(* Logix 5000 project; controller ODSI_Testing vendor 1 type 14 code 151 rev 20.19; software revision 20.05; part 2 of 2 *)
(* tags used below, declared in another part *)
   HMI_Stop_B9 : BOOL;   // Stop PB on HMI
   ODSI_Fail_Sample1_B9 : ALIAS FOR Local:6:I.Data.8;   // ODSI sent a fail signal for sample 1
   ODSI_Fail_Sample2_B9 : ALIAS FOR Local:6:I.Data.10;   // ODSI sent a fail signal for sample 2
   ODSI_Fail_Sample3_B9 : ALIAS FOR Local:6:I.Data.12;   // ODSI sent a fail signal for sample 3
   ODSI_Pass_Sample1_B9 : ALIAS FOR Local:6:I.Data.7;   // ODSI sent a pass signal for sample 1
   ODSI_Pass_Sample2_B9 : ALIAS FOR Local:6:I.Data.9;   // ODSI sent a pass signal for sample 2
   ODSI_Pass_Sample3_B9 : ALIAS FOR Local:6:I.Data.11;   // ODSI sent a pass signal for sample 3
   ODSI_Valve1_B9 : ALIAS FOR Local:6:I.Data.4;   // ODSI requests to open valve 1
   ODSI_Valve2_B9 : ALIAS FOR Local:6:I.Data.5;   // ODSI requests to open valve 2
   ODSI_Valve3_B9 : ALIAS FOR Local:6:I.Data.6;   // ODSI requests to open valve 3
   RandomDelay : DINT;   // Random number generator 0-19
   RNG_Delay_Active_B9 : BOOL;   // HMI PB randomizing valve open delay
   S1_B9_10s_Timer : TIMER;   // Releases "ACQC in" signal after 10 seconds
   S1_PB_Input_B9 : BOOL;   // HMI PB requesting sample 1
   S1_Request_B9 : ALIAS FOR Local:5:O.Data.8;   // Output to ODSI to request Sample 1
   S2_B9_10s_Timer : TIMER;   // Releases "ACQC in" signal after 10 seconds
   S2_PB_Input_B9 : BOOL;   // HMI PB requesting sample 2
   S2_Request_B9 : ALIAS FOR Local:5:O.Data.9;   // Output to ODSI to request Sample 2
   S3_B9_10s_Timer : TIMER;   // Releases "ACQC in" signal after 10 seconds
   S3_PB_Input_B9 : BOOL;   // HMI PB requesting sample 3
   S3_Request_B9 : ALIAS FOR Local:5:O.Data.10;   // Output to ODSI to request Sample 3
   System_Running_B9 : ALIAS FOR Local:6:I.Data.3;   // ODSI signal that indicates the system is currently analyzing a sample
   Valve1_Open_B9 : ALIAS FOR Local:5:O.Data.11;   // Output to ODSI confirming valve 1 is open
   Valve1_Open_Delay_B9 : TIMER;   // Delay after Request is Initiated from ODSI
   Valve1_Open_Random_Delay_B9 : TIMER;   // Randomized delay after request for valve position is received from ODSI
   Valve2_Open_B9 : ALIAS FOR Local:5:O.Data.12;   // Output to ODSI confirming valve 2 is open
   Valve2_Open_Delay_B9 : TIMER;   // Delay after Request is Initiated from ODSI
   Valve2_Open_Random_Delay_B9 : TIMER;   // Randomized delay after request for valve position is received from ODSI
   Valve3_Open_B9 : ALIAS FOR Local:5:O.Data.13;   // Output to ODSI confirming valve 3 is open
   Valve3_Open_Delay_B9 : TIMER;   // Delay after Request is Initiated from ODSI
   Valve3_Open_Random_Delay_B9 : TIMER;   // Randomized delay after request for valve position is received from ODSI
   Valve_Block_B9 : BOOL;   // HMI PB to prevent valves from opening
   Valve_Delay_B9 : DINT;
(* MainProgram, continued *)

ROUTINE Remote_B9   (* ladder *)
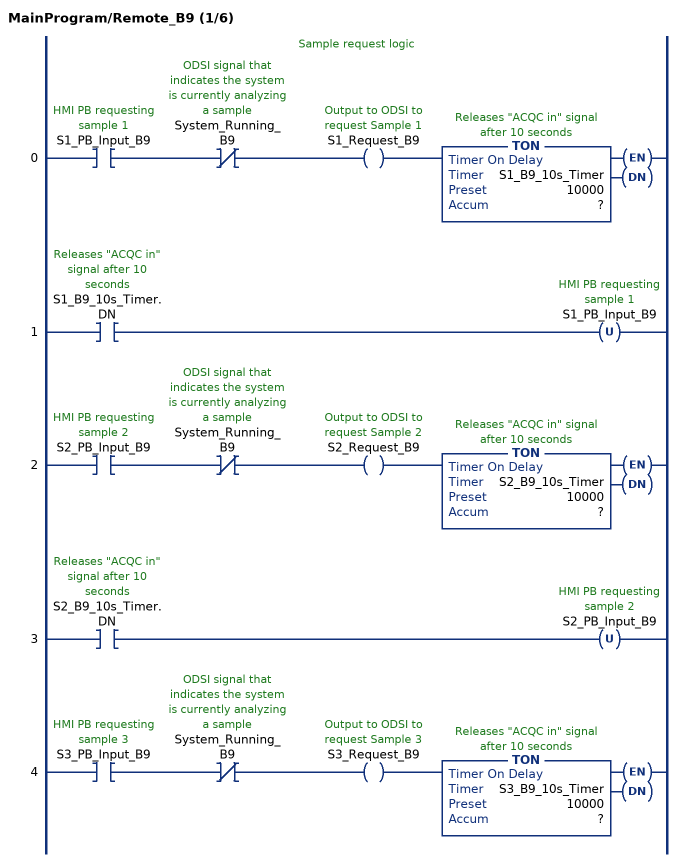
   // Sample request logic
   0: XIC(S1_PB_Input_B9)XIO(System_Running_B9)OTE(S1_Request_B9)TON(S1_B9_10s_Timer,?,?);
   1: XIC(S1_B9_10s_Timer.DN)OTU(S1_PB_Input_B9);
   2: XIC(S2_PB_Input_B9)XIO(System_Running_B9)OTE(S2_Request_B9)TON(S2_B9_10s_Timer,?,?);
   3: XIC(S2_B9_10s_Timer.DN)OTU(S2_PB_Input_B9);
   4: XIC(S3_PB_Input_B9)XIO(System_Running_B9)OTE(S3_Request_B9)TON(S3_B9_10s_Timer,?,?);
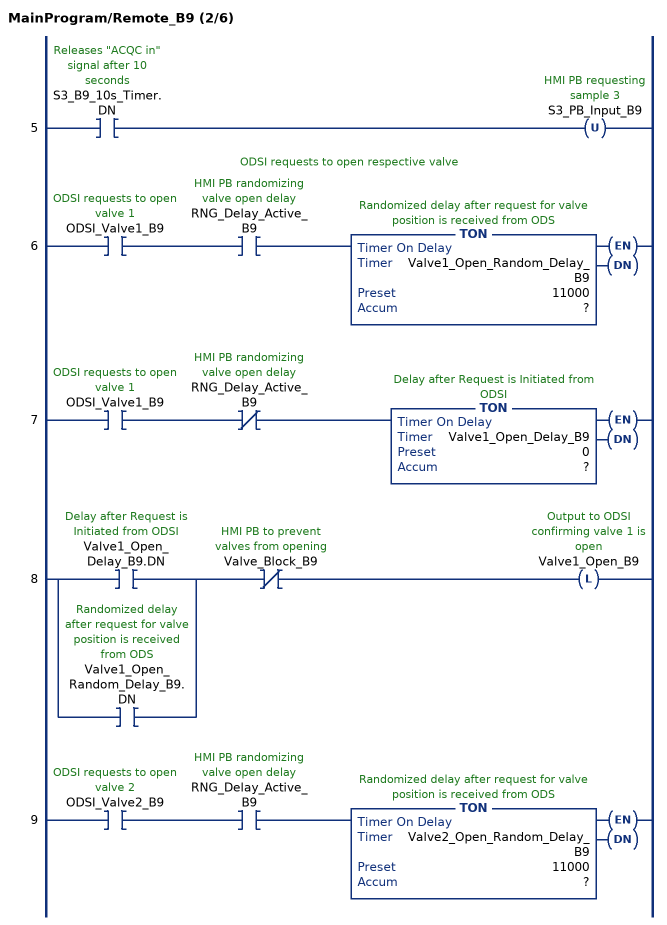
   5: XIC(S3_B9_10s_Timer.DN)OTU(S3_PB_Input_B9);
   // ODSI requests to open respective valve
   6: XIC(ODSI_Valve1_B9)XIC(RNG_Delay_Active_B9)TON(Valve1_Open_Random_Delay_B9,?,?);
   7: XIC(ODSI_Valve1_B9)XIO(RNG_Delay_Active_B9)TON(Valve1_Open_Delay_B9,?,?);
   8: [XIC(Valve1_Open_Delay_B9.DN) ,XIC(Valve1_Open_Random_Delay_B9.DN) ]XIO(Valve_Block_B9)OTL(Valve1_Open_B9);
   9: XIC(ODSI_Valve2_B9)XIC(RNG_Delay_Active_B9)TON(Valve2_Open_Random_Delay_B9,?,?);
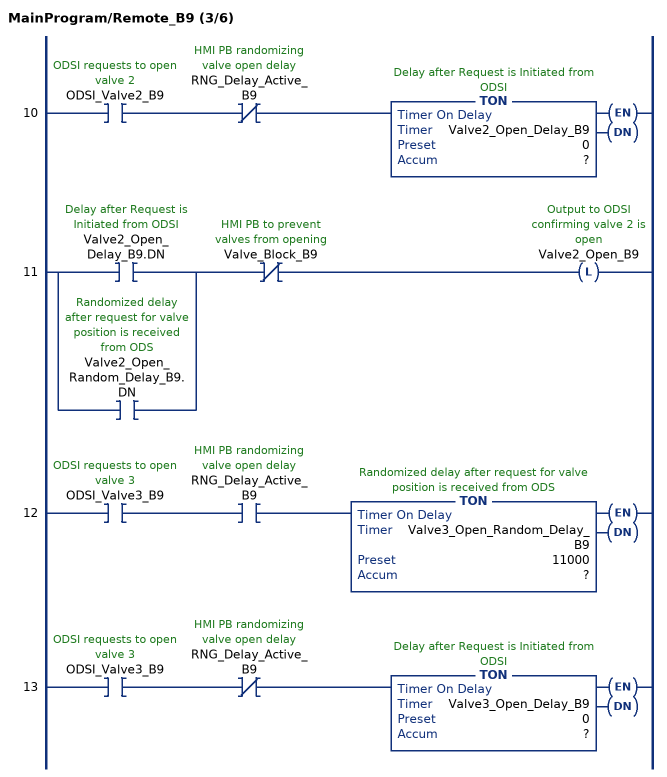
   10: XIC(ODSI_Valve2_B9)XIO(RNG_Delay_Active_B9)TON(Valve2_Open_Delay_B9,?,?);
   11: [XIC(Valve2_Open_Delay_B9.DN) ,XIC(Valve2_Open_Random_Delay_B9.DN) ]XIO(Valve_Block_B9)OTL(Valve2_Open_B9);
   12: XIC(ODSI_Valve3_B9)XIC(RNG_Delay_Active_B9)TON(Valve3_Open_Random_Delay_B9,?,?);
   13: XIC(ODSI_Valve3_B9)XIO(RNG_Delay_Active_B9)TON(Valve3_Open_Delay_B9,?,?);
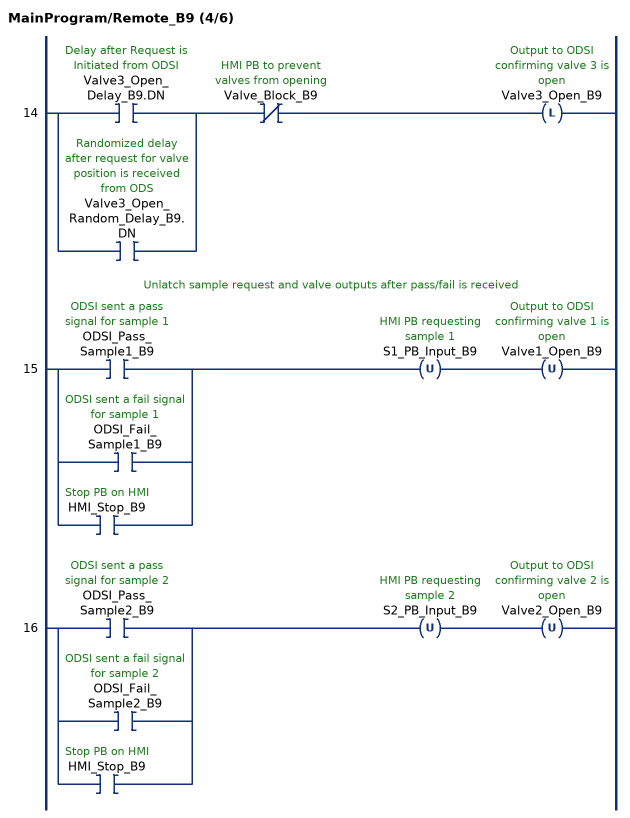
   14: [XIC(Valve3_Open_Delay_B9.DN) ,XIC(Valve3_Open_Random_Delay_B9.DN) ]XIO(Valve_Block_B9)OTL(Valve3_Open_B9);
   // Unlatch sample request and valve outputs after pass/fail is received
   15: [XIC(ODSI_Pass_Sample1_B9) ,XIC(ODSI_Fail_Sample1_B9) ,XIC(HMI_Stop_B9) ]OTU(S1_PB_Input_B9)OTU(Valve1_Open_B9);
   16: [XIC(ODSI_Pass_Sample2_B9) ,XIC(ODSI_Fail_Sample2_B9) ,XIC(HMI_Stop_B9) ]OTU(S2_PB_Input_B9)OTU(Valve2_Open_B9);
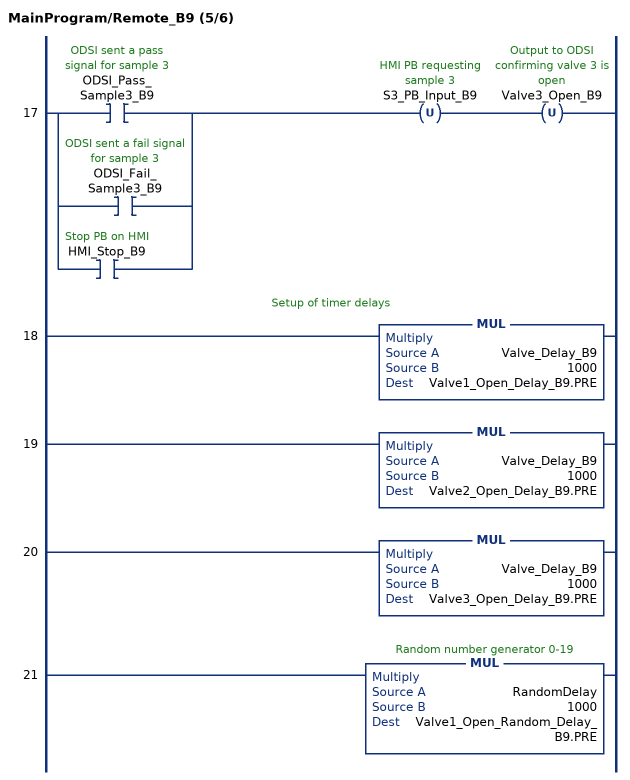
   17: [XIC(ODSI_Pass_Sample3_B9) ,XIC(ODSI_Fail_Sample3_B9) ,XIC(HMI_Stop_B9) ]OTU(S3_PB_Input_B9)OTU(Valve3_Open_B9);
   // Setup of timer delays
   18: MUL(Valve_Delay_B9,1000,Valve1_Open_Delay_B9.PRE);
   19: MUL(Valve_Delay_B9,1000,Valve2_Open_Delay_B9.PRE);
   20: MUL(Valve_Delay_B9,1000,Valve3_Open_Delay_B9.PRE);
   21: MUL(RandomDelay,1000,Valve1_Open_Random_Delay_B9.PRE);
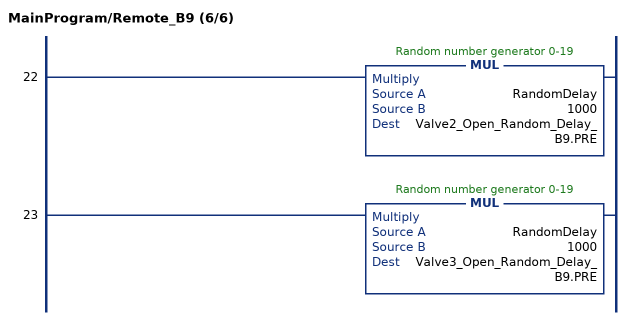
   22: MUL(RandomDelay,1000,Valve2_Open_Random_Delay_B9.PRE);
   23: MUL(RandomDelay,1000,Valve3_Open_Random_Delay_B9.PRE);
END_ROUTINE
END_PROGRAM
